FUNCTION_BLOCK Timer_TON (* Composite Function Block Type *)
  (* Standard: 61499-2 *)
  (* Version 0.0, 5/24/2016, gulzha, nxtControl GmbH, template *)
  PACKAGE Main;
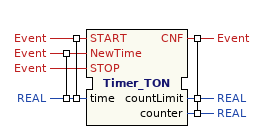
  EVENT_INPUT
    START WITH time; (* Begin Delay *)
    NewTime WITH time;
    STOP; (* Cancel Delay *)
  END_EVENT
  EVENT_OUTPUT
    CNF WITH countLimit, counter; (* Execution Confirmation *)
  END_EVENT
  VAR_INPUT
    time : REAL;
  END_VAR
  VAR_OUTPUT
    countLimit : REAL;
    counter : REAL;
  END_VAR
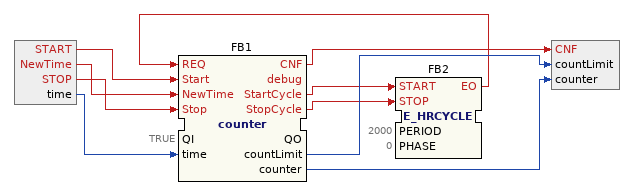
  FBS
    FB2 : E_HRCYCLE(PERIOD := 2000, PHASE := 0);
    FB1 : counter(QI := TRUE);
  END_FBS
  EVENT_CONNECTIONS
    NewTime TO FB1.NewTime;
    FB1.CNF TO CNF;
    STOP TO FB1.Stop;
    START TO FB1.Start;
    FB2.EO TO FB1.REQ;
    FB1.StartCycle TO FB2.START;
    FB1.StopCycle TO FB2.STOP;
  END_CONNECTIONS
  DATA_CONNECTIONS
    time TO FB1.time;
    FB1.countLimit TO countLimit;
    FB1.counter TO counter;
  END_CONNECTIONS
END_FUNCTION_BLOCK
